FUNCTION_BLOCK AND (* Basic Function Block Type *)
  (* Standard: 61499-2 *)
  (* Version 0.2, 2003-12-04, JHC, Rockwell Automation, Renamed for better indexing. *)
  (* Version 0.1, 2002-11-05, JHC, Rockwell Automation, Corrected missing ST element in Algorithm REQ. *)
  (* Version 0.0, 2000-05-30, JHC, Rockwell Automation *)
  (* Compiler header: package fb.rt.pnp; *)
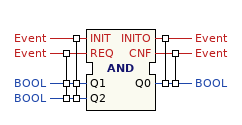
  EVENT_INPUT
    INIT WITH Q1, Q2; (* Initialization Request *)
    REQ WITH Q1, Q2; (* Normal Execution Request *)
  END_EVENT
  EVENT_OUTPUT
    INITO WITH Q0; (* Initialization Confirm *)
    CNF WITH Q0; (* Execution Confirmation *)
  END_EVENT
  VAR_INPUT
    Q1 : BOOL; (* Input event qualifier *)
    Q2 : BOOL;
  END_VAR
  VAR_OUTPUT
    Q0 : BOOL; (* Output event qualifier *)
  END_VAR
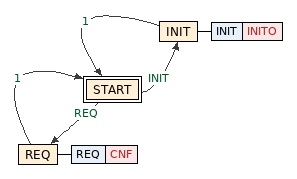
  EC_STATES
    START; (* Initial State *)
    INIT : INIT -> INITO; (* Initialization *)
    REQ : REQ -> CNF; (* Normal execution *)
  END_STATES
  EC_TRANSITIONS
    START TO INIT := INIT;
    INIT TO START := 1;
    START TO REQ := REQ;
    REQ TO START := 1;
  END_TRANSITIONS
  ALGORITHM INIT IN Java: (* Initialization algorithm *)
Q0.value=Q1.value&Q2.value;
  END_ALGORITHM
  ALGORITHM REQ IN Java: (* Normally executed algorithm *)
Q0.value=Q1.value&Q2.value;
  END_ALGORITHM
END_FUNCTION_BLOCK
